FUNCTION_BLOCK xPlanarUtility
VAR_INPUT
END_VAR
VAR_OUTPUT
END_VAR
VAR
	Running			: BYTE;	

	i				: BYTE;
	MoverEnabled	: ARRAY [1..xPlanarLink.MoverCount] OF BOOL;
	MoverInError	: ARRAY [1..xPlanarLink.MoverCount] OF BOOL;
	MoverBusy		: ARRAY [1..xPlanarLink.MoverCount] OF BOOL;
	MoverDone		: Array [1..xPlanarLink.MoverCount] OF BOOL;
END_VAR


Running := Running + 1;

UpdateObject();

ReadStatus();

METHOD ReadStatus : BOOL
VAR_INPUT
END_VAR

FOR i := 1 TO xPlanarLink.MoverCount DO
	
	IF xPlanarLink.PlanarMover[i].MCTOPLC.STD.State = 3 THEN
		MoverEnabled[i] := TRUE;
	ELSE
		MoverEnabled[i] := FALSE;
	END_IF
	
	MoverInError[i] := xPlanarLink.PlanarFeedback[i].Error;
	
	MoverBusy[i] := xPlanarLink.PlanarFeedback[i].Busy;
	
	MoverDone[i] := xPlanarLink.PlanarFeedback[i].Done;
	
END_FOR
END_METHOD

METHOD UpdateObject : BOOL
VAR_INPUT
END_VAR

FOR i := 1 TO xPlanarLink.MoverCount DO
	xPlanarLink.PlanarMover[i].Update();
	xPlanarLink.PlanarFeedback[i].Update();
END_FOR
END_METHOD

END_FUNCTION_BLOCK

(* stored: Version 1.1.0.1, ProductVersion 3.1.4024.12
   POU xPlanarUtility: Id {275caf48-8ada-48c8-87c5-223e20d4cd4a}, SpecialFunc None
   Method ReadStatus: Id {232dbaf6-8115-48c1-9a63-e2b1a144d824}
   Method UpdateObject: Id {27b8a20c-c40d-4aae-ae59-bfc6ede242c6} *)
